INTERFACE I_DriveDouble EXTENDS I_Drive

METHOD SwitchReverseOff : BOOL
VAR_INPUT
END_VAR
END_METHOD

METHOD SwitchReverseOn : BOOL
VAR_INPUT
END_VAR
END_METHOD

END_INTERFACE

(* stored: Version 1.1.0.1, ProductVersion 3.1.4024.12
   Itf I_DriveDouble: Id {1898bbb9-7de6-4ade-a5ba-272ca7e8becb}
   Method SwitchReverseOff: Id {1555693e-a721-42b9-8198-c8149cd8a3a7}
   Method SwitchReverseOn: Id {a6680044-004f-4e62-a40e-bf6860aaccbf} *)
